KUKA KRL data list: e_fraes2.dat

&ACCESS RVP1
&REL 1
&COMMENT Fresa X1
&PARAM TEMPLATE = C:\KRC\Roboter\Template\vorgabe
&PARAM EDITMASK = *
DEFDAT  E_FRAES2
;FOLD EXTERNAL DECLARATIONS;%{PE}%V3.2.0,%MKUKATPBASIS,%CEXT,%VCOMMON,%P
;FOLD BAS EXT;%{PE}%V3.2.0,%MKUKATPBASIS,%CEXT,%VEXT,%P
EXT  BAS (BAS_COMMAND  :IN,REAL  :IN )
DECL INT SUCCESS
;ENDFOLD
;FOLD A10 EXT;%{E}%V3.2.0,%MKUKATPARC,%CEXT,%VEXT,%P
EXT  A10 (A_CMD_T  :IN,A_STRT_T  :IN,A_WELD_T  :IN,A_END_T  :IN,INT  :IN )
;ENDFOLD
;FOLD A20 EXT;%{E}%V3.2.0,%MKUKATPA20,%CEXT,%VEXT,%P
EXT  A20 (INT  :IN,WELD_ST  :IN,WELD_FI  :IN,INT  :IN )
;ENDFOLD
;FOLD GRIPPER EXT;%{E}%V3.2.0,%MKUKATPGRIPPER,%CEXT,%VEXT,%P
EXT  H50 (INT  :IN,INT  :IN,INT  :IN,GRP_TYP  :IN )
;ENDFOLD
;FOLD SPOT EXT;%{E}%V3.2.0,%MKUKATPSPOT,%CEXT,%VEXT,%P
EXT  USERSPOT (S_COMMAND  :IN,SPOT_TYPE  :IN )
;ENDFOLD
;FOLD TOUCHSENSE EXT;%{E}%V3.2.0,%MKUKATPTS,%CEXT,%VEXT,%P
EXT  H70 (INT  :IN,SRCH_TYP_2  :OUT,E6POS  :IN,SRCH_TYP_3  :IN,SRCH_TYP_2  :IN,SRCH_TYP_2  :IN,SRCH_TYP_2  :IN,SRCH_TYP_2  :IN,SRCH_TYP_2  :IN,INT  :IN )
;ENDFOLD
;FOLD USER EXT;%{E}%V3.2.0,%MKUKATPUSER,%CEXT,%VEXT,%P
;Make here your modifications
;ENDFOLD
;ENDFOLD

DECL SPOT_SUGG_T LAST_SPOT={GUN[] "3                       ",RETR_CMD[] "#OPN                    ",CHOISE[] "#FIRST                  ",CLO_TM[] "1                       ",PGNO1[] "1                       ",PRESS1[] "0                       ",PGNO2[] "1                       ",PRESS2[] "0                       ",SPOT_PARAMS[] "NORMAL                  "}
DECL BASIS_SUGG_T LAST_BASIS={POINT1[] "pFresa_0                ",POINT2[] "pFresa_0                ",CP_PARAMS[] "CPDAT4                  ",PTP_PARAMS[] "PDAT25                  ",CONT[] "                        ",CP_VEL[] "0.35                    ",PTP_VEL[] "100                     "}
DECL E6POS XPS230R01010002={x 628.990417,y 2430.78589,z 93.4019775,a -130.689804,b 83.6311264,c 143.373306,s 6,t 51,e1 0.0,e2 0.0,e3 0.0,e4 0.0,e5 0.0,e6 0.0}
DECL FDAT FPS230R01010002={TOOL_NO 2,BASE_NO 0,IPO_FRAME #BASE}
DECL PDAT PPDAT1={VEL 100.0,ACC 100.0,APO_DIST 100.0}
DECL E6POS Xp001={x 628.990417,y 2430.78589,z 93.4019775,a -130.689804,b 83.6311264,c 143.373306,s 6,t 51,e1 0.0,e2 0.0,e3 0.0,e4 0.0,e5 0.0,e6 0.0}
DECL FDAT Fp001={TOOL_NO 2,BASE_NO 0,IPO_FRAME #BASE}
DECL FDAT FDress_x1={TOOL_NO 2,BASE_NO 0,IPO_FRAME #BASE}
DECL E6POS XDress_x1={x 935.442688,y 2431.45801,z -4.45435476,a -7.90584517,b 81.3359833,c -96.5874176,s 6,t 51,e1 0.0,e2 0.0,e3 0.0,e4 0.0,e5 0.0,e6 0.0}
DECL E6POS XPFRESA_01={x 1388.552,y 1126.62903,z 1573.04895,a 55.2709007,b -51.7002792,c 70.3624115,s 2,t 35,e1 0.0,e2 0.0,e3 0.0,e4 0.0,e5 0.0,e6 0.0}
DECL FDAT FpFresa_01={TOOL_NO 2,BASE_NO 0,IPO_FRAME #BASE}
DECL PDAT PPDAT2={VEL 100.0,ACC 100.0,APO_DIST 100.0}
DECL E6POS XPFRESA_02={x 881.144226,y 2206.8269,z 1046.28699,a 153.253693,b 3.1797359,c 90.6035919,s 2,t 35,e1 0.0,e2 0.0,e3 0.0,e4 0.0,e5 0.0,e6 0.0}
DECL FDAT FpFresa_02={TOOL_NO 2,BASE_NO 0,IPO_FRAME #BASE}
DECL PDAT PPDAT3={VEL 100.0,ACC 100.0,APO_DIST 100.0}
DECL E6POS XPFRESA_03={x 919.960388,y 2394.21899,z 117.4888,a -15.7696199,b 86.138443,c -102.699402,s 6,t 51,e1 0.0,e2 0.0,e3 0.0,e4 0.0,e5 0.0,e6 0.0}
DECL FDAT FpFresa_03={TOOL_NO 2,BASE_NO 0,IPO_FRAME #BASE}
DECL PDAT PPDAT4={VEL 100.0,ACC 100.0,APO_DIST 100.0}
DECL E6POS XPFRESA_04={x 933.890991,y 2391.86304,z -1.17514706,a -7.96984196,b 81.334343,c -96.6534729,s 6,t 51,e1 0.0,e2 0.0,e3 0.0,e4 0.0,e5 0.0,e6 0.0}
DECL FDAT FpFresa_04={TOOL_NO 2,BASE_NO 0,IPO_FRAME #BASE}
DECL LDAT LCPDAT1={VEL 2.0,ACC 100.0,APO_DIST 100.0,APO_FAC 50.0}
DECL E6POS XPFRESA_05={x 922.47052,y 2386.61401,z 11.7058601,a 172.544098,b 80.3358383,c 94.5076828,s 2,t 3,e1 0.0,e2 0.0,e3 0.0,e4 0.0,e5 0.0,e6 0.0}
DECL FDAT FpFresa_05={TOOL_NO 2,BASE_NO 0,IPO_FRAME #BASE}
DECL LDAT LCPDAT2={VEL 2.0,ACC 100.0,APO_DIST 100.0,APO_FAC 50.0}
DECL E6POS XPFRESA_06={x 953.203003,y 2374.521,z 195.592407,a -176.211807,b 79.2073135,c 107.4132,s 6,t 51,e1 0.0,e2 0.0,e3 0.0,e4 0.0,e5 0.0,e6 0.0}
DECL FDAT FpFresa_06={TOOL_NO 2,BASE_NO 0,IPO_FRAME #BASE}
DECL LDAT LCPDAT3={VEL 2.0,ACC 100.0,APO_DIST 100.0,APO_FAC 50.0}
DECL E6POS XPFRESA_07={x 775.328979,y 1838.18799,z 941.839294,a 152.792694,b 51.9504395,c 89.0040207,s 6,t 51,e1 0.0,e2 0.0,e3 0.0,e4 0.0,e5 0.0,e6 0.0}
DECL FDAT FpFresa_07={TOOL_NO 2,BASE_NO 0,IPO_FRAME #BASE}
DECL PDAT PPDAT5={VEL 100.0,ACC 100.0,APO_DIST 100.0}
DECL E6POS XPFRESA_08={x 939.487305,y 1800.54797,z 2203.9541,a 128.640503,b -23.3977604,c 36.4649696,s 2,t 3,e1 0.0,e2 0.0,e3 0.0,e4 0.0,e5 0.0,e6 0.0}
DECL FDAT FpFresa_08={TOOL_NO 2,BASE_NO 0,IPO_FRAME #BASE}
DECL PDAT PPDAT6={VEL 100.0,ACC 100.0,APO_DIST 100.0}
DECL E6POS XPSOLDAX1={x 644.040283,y 2430.77588,z 104.992104,a -100.702698,b 85.9585419,c 169.755798,s 6,t 51,e1 0.0,e2 0.0,e3 0.0,e4 0.0,e5 0.0,e6 0.0}
DECL FDAT FpSoldaX1={TOOL_NO 2,BASE_NO 0,IPO_FRAME #BASE}
DECL PDAT PPDAT7={VEL 100.0,ACC 100.0,APO_DIST 100.0}
DECL FDAT FDress_x={TOOL_NO 2,BASE_NO 0,IPO_FRAME #BASE}
DECL E6POS XDress_x={x 644.040283,y 2430.77588,z 104.992104,a -100.702698,b 85.9585419,c 169.755798,s 6,t 51,e1 0.0,e2 0.0,e3 0.0,e4 0.0,e5 0.0,e6 0.0}
DECL E6POS XPSOLDAX={x 1658.10999,y -21.3289509,z 728.15332,a -34.7539291,b -3.29387903,c 121.445297,s 2,t 3,e1 0.0,e2 0.0,e3 0.0,e4 0.0,e5 0.0,e6 0.0}
DECL FDAT FpSoldaX={TOOL_NO 2,BASE_NO 0,IPO_FRAME #BASE}
DECL LDAT LCPDAT4={VEL 2.0,ACC 100.0,APO_DIST 100.0,APO_FAC 50.0}
DECL PDAT PPDAT8={VEL 50.0,ACC 100.0,APO_DIST 100.0}
DECL PDAT PPDAT9={VEL 100.0,ACC 100.0,APO_DIST 10.0}
DECL PDAT PPDAT10={VEL 100.0,ACC 100.0,APO_DIST 10.0}
DECL PDAT PPDAT11={VEL 100.0,ACC 100.0,APO_DIST 10.0}
DECL PDAT PPDAT12={VEL 100.0,ACC 100.0,APO_DIST 10.0}
DECL PDAT PPDAT13={VEL 100.0,ACC 100.0,APO_DIST 10.0}
DECL PDAT PPDAT14={VEL 100.0,ACC 100.0,APO_DIST 10.0}
DECL PDAT PPDAT15={VEL 100.0,ACC 100.0,APO_DIST 10.0}
DECL PDAT PPDAT16={VEL 100.0,ACC 100.0,APO_DIST 10.0}
DECL LDAT LCPDAT5={VEL 2.0,ACC 100.0,APO_DIST 100.0,APO_FAC 50.0}
DECL E6POS XPFRESA_4={x 898.384827,y 2309.20093,z 210.289795,a 165.421204,b 68.3341064,c 83.9502411,s 2,t 3,e1 0.0,e2 0.0,e3 0.0,e4 0.0,e5 0.0,e6 0.0}
DECL FDAT FpFresa_4={TOOL_NO 2,BASE_NO 0,IPO_FRAME #BASE}
DECL PDAT PPDAT17={VEL 100.0,ACC 100.0,APO_DIST 10.0}
DECL PDAT PPDAT18={VEL 100.0,ACC 100.0,APO_DIST 10.0}
DECL PDAT PPDAT19={VEL 100.0,ACC 100.0,APO_DIST 10.0}
DECL PDAT PPDAT20={VEL 100.0,ACC 100.0,APO_DIST 10.0}
DECL E6POS XPFRESA_3={x 898.362488,y 2309.18994,z 210.282303,a 165.423904,b 68.3332672,c 83.9527969,s 2,t 3,e1 0.0,e2 0.0,e3 0.0,e4 0.0,e5 0.0,e6 0.0}
DECL FDAT FpFresa_3={TOOL_NO 2,BASE_NO 0,IPO_FRAME #BASE}
DECL PDAT PPDAT21={VEL 100.0,ACC 100.0,APO_DIST 10.0}
DECL PDAT PPDAT22={VEL 100.0,ACC 100.0,APO_DIST 10.0}
DECL PDAT PPDAT23={VEL 100.0,ACC 100.0,APO_DIST 10.0}
DECL E6POS XPFRESA_0={x 1658.10205,y -21.3623295,z 728.221313,a -34.7549706,b -3.29463005,c 121.444801,s 2,t 3,e1 0.0,e2 0.0,e3 0.0,e4 0.0,e5 0.0,e6 0.0}
DECL FDAT FpFresa_0={TOOL_NO 2,BASE_NO 0,IPO_FRAME #BASE}
DECL PDAT PPDAT24={VEL 100.0,ACC 100.0,APO_DIST 10.0}
DECL PDAT PPDAT25={VEL 100.0,ACC 100.0,APO_DIST 10.0}
DECL E6POS XpSoldaX2={x 919.983582,y 2394.22998,z 117.436699,a -15.7574701,b 86.1378021,c -102.6866,s 6,t 51,e1 0.0,e2 0.0,e3 0.0,e4 0.0,e5 0.0,e6 0.0}
DECL FDAT FpSoldaX2={TOOL_NO 2,BASE_NO 0,IPO_FRAME #BASE}
DECL PDAT PPDAT26={VEL 50.0,ACC 100.0,APO_DIST 100.0}
DECL SPOT_TYPE SNORMAL
DECL E6POS XpSoldaX3={x 919.960388,y 2394.21899,z 117.4888,a -15.7696199,b 86.138443,c -102.699402,s 6,t 51,e1 0.0,e2 0.0,e3 0.0,e4 0.0,e5 0.0,e6 0.0}
DECL FDAT FpSoldaX3={TOOL_NO 2,BASE_NO 0,IPO_FRAME #BASE}
DECL PDAT PPDAT27={VEL 50.0,ACC 100.0,APO_DIST 100.0}
ENDDAT
